// Mitsubishi GX Works2 project: 42015016   PLC: Q00J
// 42015016

PROGRAM MAIN
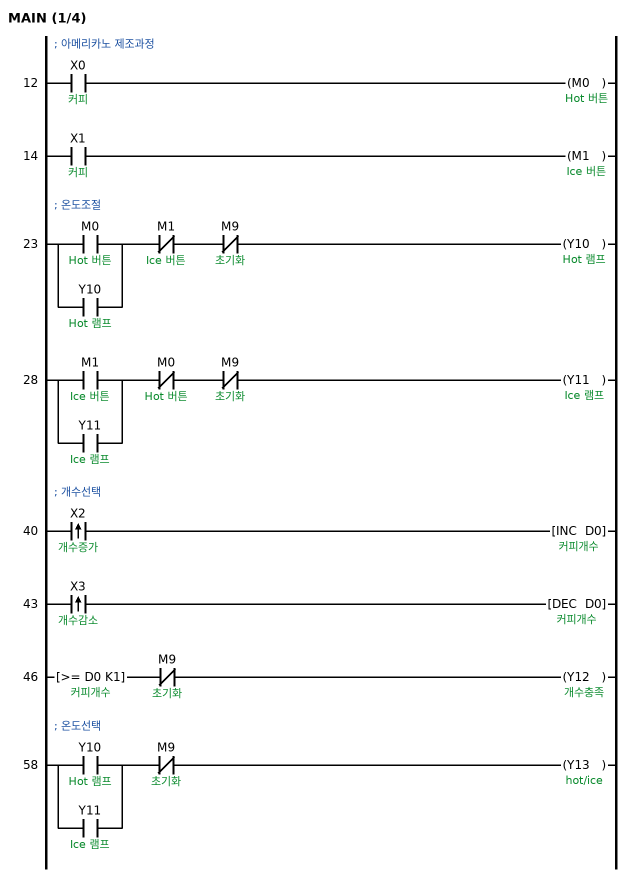
; 아메리카노 제조과정
12    LD      X0  ; 커피
      OUT     M0  ; Hot 버튼
14    LD      X1  ; 커피
      OUT     M1  ; Ice 버튼
; 온도조절
23    LD      M0  ; Hot 버튼
      OR      Y10  ; Hot 램프
      ANI     M1  ; Ice 버튼
      ANI     M9  ; 초기화
      OUT     Y10  ; Hot 램프
28    LD      M1  ; Ice 버튼
      OR      Y11  ; Ice 램프
      ANI     M0  ; Hot 버튼
      ANI     M9  ; 초기화
      OUT     Y11  ; Ice 램프
; 개수선택
40    LDP     X2  ; 개수증가
      INC     D0  ; 커피개수
43    LDP     X3  ; 개수감소
      DEC     D0
46    LD>=    D0 K1  ; 커피개수
      ANI     M9  ; 초기화
      OUT     Y12  ; 개수충족
; 온도선택
58    LD      Y10  ; Hot 램프
      OR      Y11  ; Ice 램프
      ANI     M9  ; 초기화
      OUT     Y13  ; hot/ice
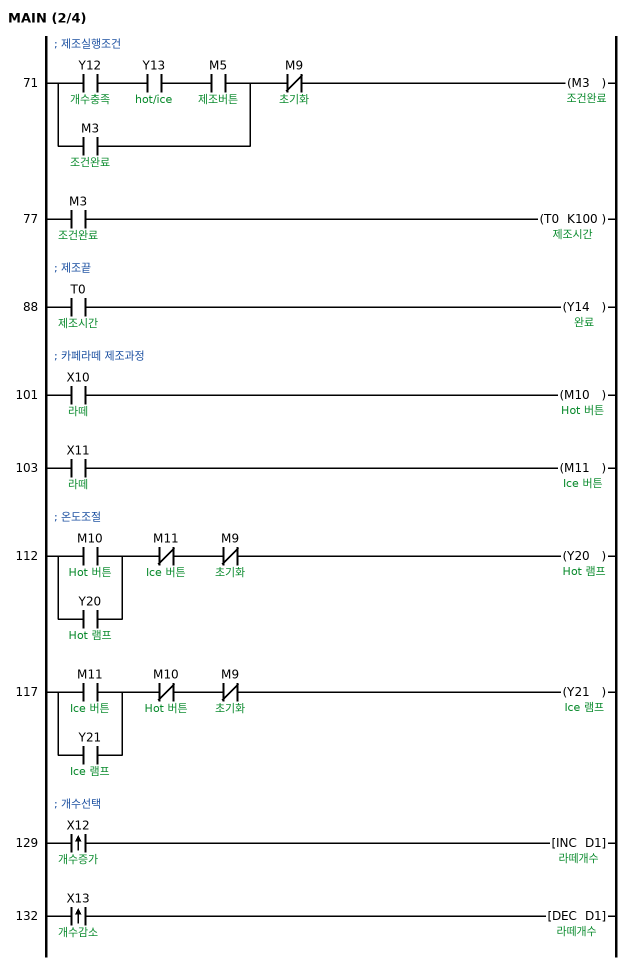
; 제조실행조건
71    LD      Y12  ; 개수충족
      AND     Y13  ; hot/ice
      AND     M5  ; 제조버튼
      OR      M3  ; 조건완료
      ANI     M9  ; 초기화
      OUT     M3  ; 조건완료
77    LD      M3  ; 조건완료
      OUT     T0 K100  ; 제조시간
; 제조끝
88    LD      T0  ; 제조시간
      OUT     Y14  ; 완료
; 카페라떼 제조과정
101   LD      X10  ; 라떼
      OUT     M10  ; Hot 버튼
103   LD      X11  ; 라떼
      OUT     M11  ; Ice 버튼
; 온도조절
112   LD      M10  ; Hot 버튼
      OR      Y20  ; Hot 램프
      ANI     M11  ; Ice 버튼
      ANI     M9  ; 초기화
      OUT     Y20  ; Hot 램프
117   LD      M11  ; Ice 버튼
      OR      Y21  ; Ice 램프
      ANI     M10  ; Hot 버튼
      ANI     M9  ; 초기화
      OUT     Y21  ; Ice 램프
; 개수선택
129   LDP     X12  ; 개수증가
      INC     D1  ; 라떼개수
132   LDP     X13  ; 개수감소
      DEC     D1
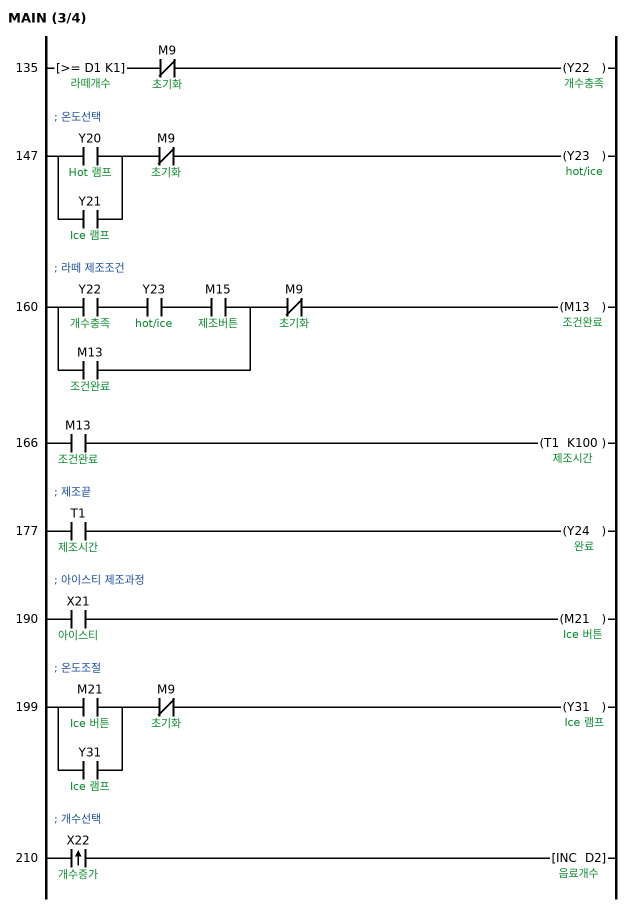
135   LD>=    D1 K1  ; 라떼개수
      ANI     M9  ; 초기화
      OUT     Y22  ; 개수충족
; 온도선택
147   LD      Y20  ; Hot 램프
      OR      Y21  ; Ice 램프
      ANI     M9  ; 초기화
      OUT     Y23  ; hot/ice
; 라떼 제조조건
160   LD      Y22  ; 개수충족
      AND     Y23  ; hot/ice
      AND     M15  ; 제조버튼
      OR      M13  ; 조건완료
      ANI     M9  ; 초기화
      OUT     M13  ; 조건완료
166   LD      M13  ; 조건완료
      OUT     T1 K100  ; 제조시간
; 제조끝
177   LD      T1  ; 제조시간
      OUT     Y24  ; 완료
; 아이스티 제조과정
190   LD      X21  ; 아이스티
      OUT     M21  ; Ice 버튼
; 온도조절
199   LD      M21  ; Ice 버튼
      OR      Y31  ; Ice 램프
      ANI     M9  ; 초기화
      OUT     Y31  ; Ice 램프
; 개수선택
210   LDP     X22  ; 개수증가
      INC     D2  ; 음료개수
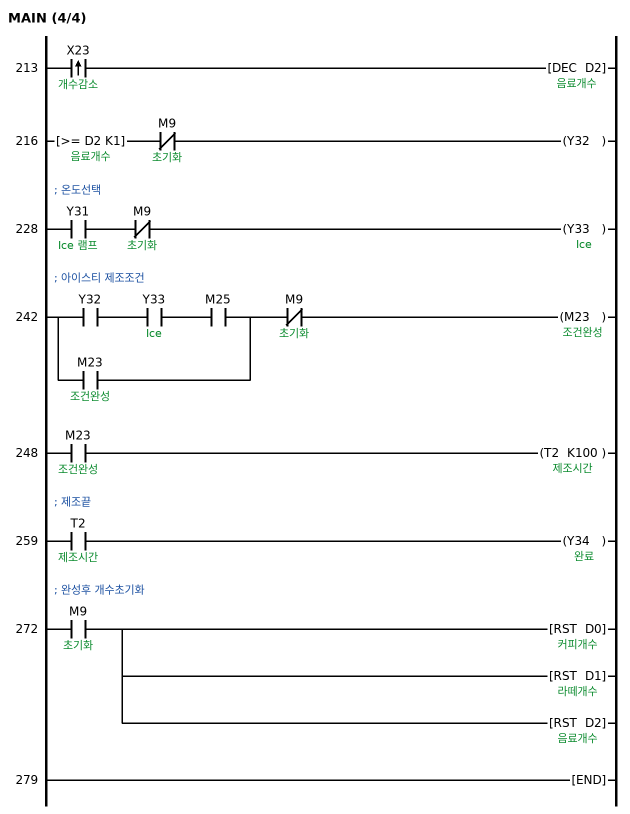
213   LDP     X23  ; 개수감소
      DEC     D2
216   LD>=    D2 K1  ; 음료개수
      ANI     M9  ; 초기화
      OUT     Y32
; 온도선택
228   LD      Y31  ; Ice 램프
      ANI     M9  ; 초기화
      OUT     Y33  ; Ice
; 아이스티 제조조건
242   LD      Y32
      AND     Y33  ; Ice
      AND     M25
      OR      M23  ; 조건완성
      ANI     M9  ; 초기화
      OUT     M23  ; 조건완성
248   LD      M23  ; 조건완성
      OUT     T2 K100  ; 제조시간
; 제조끝
259   LD      T2  ; 제조시간
      OUT     Y34  ; 완료
; 완성후 개수초기화
272   LD      M9  ; 초기화
      RST     D0  ; 커피개수
      RST     D1  ; 라떼개수
      RST     D2  ; 음료개수
279   END
END_PROGRAM
